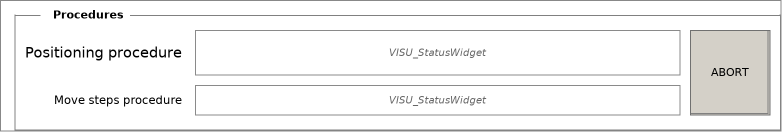
VISUALIZATION VISU_M2Procedures  // 782x132
VAR_IN_OUT
	ref : M2;
    widget : M2Widget;
END_VAR
    Polyline (130,15) (780,15) (780,130) (15,130) (15,15) (40,15)
    Frame (195,30 485x45)
        shows VISU_StatusWidget(widget := widget.movePosition.actualStatus)
    Frame (195,85 485x30)
        shows VISU_StatusWidget(widget := widget.moveSteps.actualStatus)
    Label (10,35 175x35), "Positioning procedure"
    Label (20,85 165x30), "Move steps procedure"
    Button (690,30 80x85), "ABORT", input disabled if: ref.processes.abort.statuses.enabledStatus.disabled
        OnMouseClick: execute { ref.processes.abort.do_request := TRUE; }
    Label (50,5 85x20), "Procedures"
END_VISUALIZATION

(* stored: Version 1.1.0.1, ProductVersion 3.1.4019.2
   Visu VISU_M2Procedures: Id {d2eba28d-b850-47dd-a504-0cf09c4c6373} *)
